Universal Robots PolyScope program: andrea3.urp

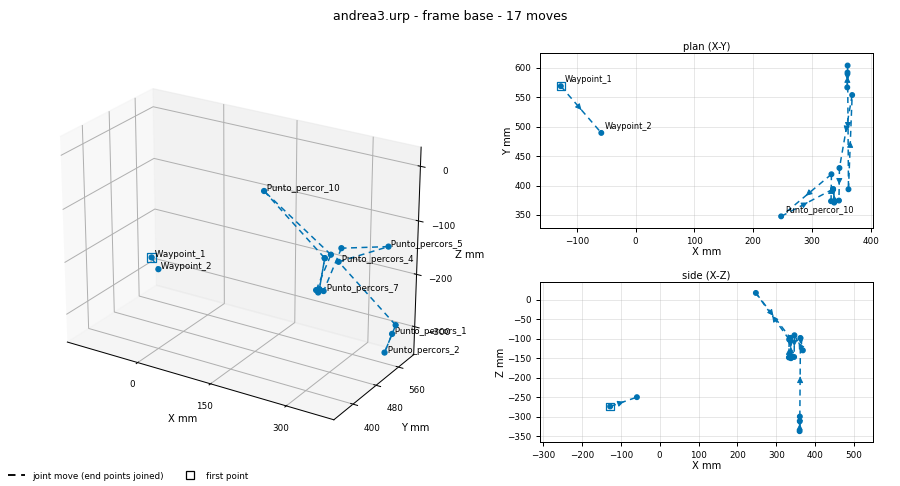
[picture p0: tool path of andrea3.urp in frame base, 17 of 20 moves have a stored position in this frame; points joined in program order, loops and branches not executed]
Program andrea3 (installation=Kong_install directory=/programs/usbdisk/andrea_mk2 createdIn=3.15.4.106291 lastSavedIn=3.15.4.106291 robotSerialNumber=2017357596)
Calibrated DH parameters: a=[0.000104, -0.381245, -0.385946, 0.00002, 0.000083, 0]; d=[0.089177, 59.99214, -36.297918, -23.584132, 0.094784, 0.082552]; alpha=[1.570197, -0.003145, 0.002952, 1.570494, -1.570091, 0]; deltaTheta=[-0.00001, -0.459739, 0.638868, -0.17972, -0.000006, -0.000462]
InitVariablesNode variables(variable(name=XY, expression=[0,0]), variable(name=countNFC, expression=0))
Robot Program (runOnlyOnce=false)
  Script file /home/ur/ursim-current/programs/relPose.script
    | def relPose(FeaturePose,vect):
    | 
    |     # FeaturePose is the pose for the feature
    |     # vect = p[0.1, 0, 0, 0, 0, 0] makes us move 10cm in the X direction of the feature
    |     # credits: https://forum.universal-robots.com/t/move-tcp-relative-to-feature/15492
    | 
    |    PoseRelativeToFeature = pose_trans(pose_inv(FeaturePose), get_actual_tcp_pose())
    |    MoveTCPRelativeToFeature = pose_add(PoseRelativeToFeature, vect)
    |    return pose_trans(FeaturePose, MoveTCPRelativeToFeature)
    | 
    | end
  Script file /home/ur/ursim-current/programs/andrea_mk2/calcPallPos1XY.script
    | def calcPallPos1XY(nPosX,distX,nPosY,distY,nPezzo):
    | 
    |     # calcola posizione del prossimo pezzo sul pallet in X e Y dal primo pezzo della griglia (origine, ossia in basso a sinistra)
    | 
    |     # nPosX è il numero di colonne
    |     # nPosY è il numero di righe
    |     # distX è la distanza tra colonne
    |     # distY è la distanza tra righe
    | 
    |     posX = nPezzo%nPosX
    |     if(posX==0): posX = 4 end
    |     posY = ceil(nPezzo/nPosX)
    | 
    |     X=distX*(posX - 1)
    |     Y=distY*(posY - 1)
    |     xy=[X,Y]
    | 
    |     return xy
    | 
    |  end
  countNFC := countNFC+1
  MoveJ speed 60 deg/s, acceleration 80 deg/s^2 (useActiveTCP=false) tcp=Ventosa
    Waypoint Waypoint_1: TCP in base x=-127.249 y=569.007 z=-273.97 mm, rx=-2.3039 ry=-0.5206 rz=-0.2288 rad; joints [-88.999, -25.01, 79.358, -9.678, 91.456, 155.199] deg; flange x=-120.447 y=603.545 z=-174.923 mm, rx=-2.3039 ry=-0.5206 rz=-0.2288 rad
  XY := calcPallPos1XY(4,18,10,8,countNFC)
  MoveJ speed 60 deg/s, acceleration 80 deg/s^2 (useActiveTCP=false) tcp=Ventosa
    SuppressedNode
      Popup Message (haltProgram=false inputType=Variable) variable=XY
    Waypoint Waypoint_2: TCP in base x=-58.441 y=489.516 z=-250.08 mm, rx=-2.2888 ry=-0.6043 rz=-0.263 rad; joints [-96.49, -34.009, 98.153, -19.269, 86.152, 145.828] deg; flange x=-58.447 y=524.429 z=-150.93 mm, rx=-2.2888 ry=-0.6043 rz=-0.263 rad
    p_pall := relPose(Piano_Carrello,p[XY[0]/1000,XY[1]/1000,0.0,0.0,0.0,0.0])
    Waypoint Punto_percors (Variable): variable=p_pall
    SuppressedNode
      centro_modulo := relPose(Piano_Carrello,p[-0.05,-0.05,0.0,0.0,0.0,0.0])
    SuppressedNode
      Waypoint Punto_percors (Variable): variable=centro_modulo
    SuppressedNode
      pezzo1 := relPose(Piano_Carrello,p[-0.0275,-0.0337,0.0,0.0,0.0,0.0])
  MoveL speed 250 mm/s, acceleration 1200 mm/s^2 (useActiveTCP=false) tcp=Ventosa; feature=Base
    p_pall := relPose(Piano_Carrello,p[0.0,0.0,-0.1,0.0,0.0,0.0])
    Waypoint Punto_percors (Variable): variable=p_pall
    Popup Message (haltProgram=false message=o inputType=Text)
    p_pall := relPose(Piano_Carrello,p[0.0,0.0,+0.1,0.0,0.0,0.0])
    Waypoint Punto_percors (Variable): variable=p_pall
  MoveJ speed 60 deg/s, acceleration 80 deg/s^2 (useActiveTCP=false) tcp=Ventosa
    Waypoint Punto_percors_1: TCP in base x=360.235 y=592.133 z=-312.029 mm, rx=-2.2888 ry=-0.6043 rz=-0.263 rad; joints [-131.868, -6.111, 42.389, 16.446, 62.296, 118.284] deg; flange x=360.229 y=627.047 z=-212.879 mm, rx=-2.2888 ry=-0.6043 rz=-0.263 rad
    Waypoint Punto_percors_2: TCP in base x=359.846 y=566.873 z=-337.553 mm, rx=-2.2887 ry=-0.6044 rz=-0.2629 rad; joints [-133.35, -6.1, 47.305, 12.155, 61.413, 116.94] deg; flange x=359.84 y=601.783 z=-238.403 mm, rx=-2.2887 ry=-0.6044 rz=-0.2629 rad
    Waypoint Punto_percors_3: TCP in base x=360.405 y=604.095 z=-299.967 mm, rx=-2.2888 ry=-0.6043 rz=-0.2631 rad; joints [-131.197, -5.882, 39.639, 18.687, 62.698, 118.883] deg; flange x=360.394 y=639.008 z=-200.817 mm, rx=-2.2888 ry=-0.6043 rz=-0.2631 rad
    Waypoint Punto_percors_4: TCP in base x=361.884 y=393.627 z=-97.825 mm, rx=-2.3321 ry=-0.5975 rz=-0.2952 rad; joints [-145.924, -43.509, 87.922, 15.491, 57.335, 104.682] deg; flange x=360.373 y=432.103 z=-0.014 mm, rx=-2.3321 ry=-0.5975 rz=-0.2952 rad
  MoveJ speed 60 deg/s, acceleration 80 deg/s^2 (useActiveTCP=false) tcp=Dosatore_Colla
    Waypoint Punto_percors_5: TCP in base x=368.156 y=553.933 z=-129.773 mm, rx=-2.3872 ry=0.0262 rz=-0.0499 rad; joints [-145.925, -43.512, 87.923, 15.491, 57.335, 104.68] deg; flange x=360.385 y=432.094 z=0.008 mm, rx=-2.3321 ry=-0.5975 rz=-0.2952 rad
    Waypoint Punto_percors_6: TCP in base x=346.525 y=429.809 z=-90.901 mm, rx=2.8684 ry=-0.498 rz=0.4963 rad; joints [-130.235, -41.25, 75.1, 55.819, 112.109, 129.678] deg; flange x=294.495 y=472.211 z=74.153 mm, rx=2.8334 ry=0.2554 rz=0.398 rad
    Waypoint Punto_percors_7: TCP in base x=345.7 y=374.489 z=-146.809 mm, rx=2.8685 ry=-0.4978 rz=0.4962 rad; joints [-134.218, -41.871, 86.428, 43.5, 112.047, 125.394] deg; flange x=293.676 y=416.87 z=18.254 mm, rx=2.8335 ry=0.2556 rz=0.3979 rad
    Waypoint Punto_percors_8: TCP in base x=332.241 y=373.424 z=-148.053 mm, rx=2.8953 ry=-0.2434 rz=0.8191 rad; joints [-129.612, -46.561, 97.376, 26.024, 119.722, 116.801] deg; flange x=241.61 y=402.136 z=2.645 mm, rx=2.7481 ry=0.4942 rz=0.7142 rad
    Waypoint Punto_percors_9: TCP in base x=332.91 y=419.209 z=-101.82 mm, rx=2.8952 ry=-0.2434 rz=0.819 rad; joints [-126.246, -46.699, 88.52, 36.923, 120.408, 120.592] deg; flange x=242.285 y=447.932 z=48.879 mm, rx=2.7481 ry=0.4942 rz=0.7141 rad
  MoveJ speed 60 deg/s, acceleration 80 deg/s^2 (useActiveTCP=false) tcp=Ventosa
    Waypoint Punto_percor_10: TCP in base x=247.37 y=347.613 z=17.849 mm, rx=2.7481 ry=0.4942 rz=0.714 rad; joints [-126.247, -46.7, 88.522, 36.924, 120.406, 120.593] deg; flange x=242.286 y=447.918 z=48.877 mm, rx=2.7481 ry=0.4942 rz=0.714 rad
    Waypoint Punto_percor_11: TCP in base x=335.749 y=393.911 z=-97.703 mm, rx=-2.0353 ry=0.1912 rz=-2.0441 rad; joints [-127.274, -47.792, 108.361, -61.985, 138.312, 104.384] deg; flange x=284.356 y=456.498 z=-30.687 mm, rx=-2.0353 ry=0.1912 rz=-2.0441 rad
    Waypoint Punto_percor_12: TCP in base x=338.359 y=373.234 z=-145.029 mm, rx=-1.712 ry=0.6311 rz=-1.7722 rad; joints [-132.228, -47.414, 117.865, -75.373, 134.377, 130.604] deg; flange x=286.4 y=396.013 z=-56.536 mm, rx=-1.712 ry=0.6311 rz=-1.7722 rad
    Waypoint Punto_percor_13: TCP in base x=337.572 y=370.981 z=-149.981 mm, rx=-1.7121 ry=0.6312 rz=-1.7722 rad; joints [-132.354, -46.82, 118.144, -76.237, 134.255, 130.611] deg; flange x=285.617 y=393.768 z=-61.488 mm, rx=-1.7121 ry=0.6312 rz=-1.7722 rad
    Waypoint Punto_percor_12: TCP in base x=338.359 y=373.234 z=-145.029 mm, rx=-1.712 ry=0.6311 rz=-1.7722 rad; joints [-132.228, -47.414, 117.865, -75.373, 134.377, 130.604] deg; flange x=286.4 y=396.013 z=-56.536 mm, rx=-1.712 ry=0.6311 rz=-1.7722 rad
    Waypoint Punto_percor_14: TCP in base x=335.761 y=393.868 z=-97.693 mm, rx=-2.0353 ry=0.1912 rz=-2.0442 rad; joints [-127.277, -47.794, 108.365, -61.99, 138.314, 104.379] deg; flange x=284.372 y=456.463 z=-30.681 mm, rx=-2.0353 ry=0.1912 rz=-2.0442 rad
